TYPE Transfo :
STRUCT
    MesWarningTemp				: BOOL ;	(* Transfo Temperature warning		    *)
    MesAlarmTemp				: BOOL ;	(* Transfo Temperature Alarm		    *)
    MesAlarmGas					: BOOL ;	(* Transfo Gas Alarm			        *)
    MesAlarmOilLevel			: BOOL ;	(* Transfo Oil Level Alarm		        *)
    MesAlarmsSynthesis			: BOOL ;	(* Transfo Synthesis Alarm              *)
                                                                             
	MesAlarmCode				: WORD ;  	(* (NA) Internal Akuo AlarmCode         *)
	MesWarningCode				: WORD ; 	(* (NA) Internal Akuo WarningCode       *)
	MesEventCode				: WORD ; 	(* (NA) Internal Akuo EventCode	        *)

END_STRUCT
END_TYPE

(* stored: Version 1.1.0.1, ProductVersion 3.1.4024.6
   DUT Transfo: Id {80c4aa5e-bc2f-4ed7-957c-a680032b5aec} *)
